Staubli VAL3: PROG.pjx

--- PROG.pjx ---
Parameters version=s7.7.1 stackSize=5000 millimeterUnit=true
Program file=delete.pgx
Program file=deleteItem.pgx
Program file=delEvent.pgx
Program file=duplicate.pgx
Program file=find.pgx
Program file=findItem.pgx
Program file=findTrajItem.pgx
Program file=get.pgx
Program file=getItem.pgx
Program file=getProgItem.pgx
Program file=getSize.pgx
Program file=getSizeItem.pgx
Program file=getType.pgx
Program file=insertItem.pgx
Program file=load.pgx
Program file=loadCycle.pgx
Program file=loadPage.pgx
Program file=new.pgx
Program file=onEdit.pgx
Program file=onInsert.pgx
Program file=onProgEnd.pgx
Program file=onRun.pgx
Program file=onStart.pgx
Program file=onStop.pgx
Program file=pasteItem.pgx
Program file=save.pgx
Program file=scan_prog.pgx
Program file=scanning.pgx
Program file=selectItem.pgx
Program file=setItem.pgx
Program file=showExist.pgx
Program file=unSelectItem.pgx
Program file=write_to_file.pgx
Data file=PROG.dtx
Library alias=saveData path=Disk://saveData/saveData.pjx
Library alias=page path=Disk://kernel/template/page/page.pjx
Library alias=saveProg path=Disk://kernel/template/session/saveProg/PROG/PROG.pjx
Library alias=use path=Disk://kernel/userPage/userPage.pjx
Library alias=language path=Disk://kernel/language/language.pjx
Library alias=cycleStatus path=Disk://cycleStatus/cycleStatus.pjx
Library alias=TrajItem path=Disk://../templates/trajectory/trajectory.pjx
Library alias=sub path=Disk://instruction/SUB/SUB.pjx
Library alias=tcp path=Disk://kernel/tool/tool.pjx
Library alias=saveInputOutput path=Disk://saveInputOutput/saveInputOutput.pjx
Type name=InstrItem path=Disk://kernel/template/InstrItem/InstrItem.pjx
Type name=progItem path=Disk://kernel/template/progItem/progItem.pjx
Type name=TrajectoryItem path=Disk://kernel/template/TrajectoryItem/TrajectoryItem.pjx

--- PROG.dtx ---
num nChar = 89
num nFile = 2
progItem pEdit
  [0]
    InstrItem iEvent[2]
      [0]
        string sType = "PALLET"
        string sData = "prise"
      [1]
        string sType = "OUT"
        string sData = "bOut0>OFF AND bOut1>ON"
    string sID = "pick_place"
public string sItems
string sLine[100]
string sPathTemplate = "Disk://kernel/template/"
string sSession
string sTrajType
public string sWrite

--- delete.pgx ---
public program delete(string x_sName (dimensions=1), num x_nResult (dimensions=1))
  local string l_sItem
  local num l_nDefault
begin
  //
  // delete the select program in
  //
  if isDefined(saveProg:pProg[x_sName])
    // delete
    delete(saveProg:pProg[x_sName])
  endIf
end

--- deleteItem.pgx ---
public program deleteItem(num x_nIndex, num& x_nResult[])
  local num l_nFound
  local num l_nSize
  local num i
  local InstrItem l_sEvent
begin
  //
  // delete the selected field
  //
  call getSizeItem(l_nSize)
  l_nFound=0
  for i=0 to (l_nSize-1)
    call getItem(l_sEvent,i)
    if find(l_sEvent.sType,"#")!=-1
      l_nFound=-1
      call delEvent(i)
      i=i-1
      call getSizeItem(l_nSize)
    endIf
  endFor
  //
  // if there are no marked events delete the select one
  //
  if x_nIndex!=-1 and l_nFound==0
    call delEvent(x_nIndex)
  endIf
end

--- delEvent.pgx ---
program delEvent(num x_nIndex (dimensions=1))
begin
  // delete the item
  if size(pEdit.iEvent)>1
    delete(pEdit.iEvent[x_nIndex])
  else
    pEdit.iEvent.sType=""
    pEdit.iEvent.sData=""
  endIf
end

--- duplicate.pgx ---
public program duplicate(string x_sCopy (dimensions=1), string x_sPaste (dimensions=1), num& x_nResult[] (dimensions=1))
  local num i
  local num l_nSize
  local string l_sItem
  local bool l_bFound
begin
  //
  // return -1 if present
  //
  // create a new one
  call new(x_sPaste,i)
  // duplicate
  saveProg:pProg[x_sPaste]=saveProg:pProg[x_sCopy]
  saveProg:pProg[x_sPaste].sID=x_sPaste
end

--- find.pgx ---
public program find(string& x_sItem[] (dimensions=1), bool& x_bFound[] (dimensions=1))
  local num i
  local num l_nSize
  local string l_sEvent
begin
  // check if the item has been found
  x_bFound=isDefined(saveProg:pProg[x_sItem])
end

--- findItem.pgx ---
public program findItem(InstrItem x_iItem, num& x_nResult[], bool x_bUseSession)
// procedure
  local num i
  local num j
  local num k
  local num l_nSize
  local string l_sProgName
  local bool l_bFound
  local num l_nSizeItem
  local InstrItem l_iItem
  local num z
  local string l_sSession
  local string l_sEmpty
  local string l_sMessage
  local string l_sPath
begin
  //
  // search in all of the program the x_iItem
  //
  // check if the cycle is running or the simulation...
  //
  // mutex the resource
  //
  if !cycleStatus:bCycle and !cycleStatus:bSimulation
    setMutex(cycleStatus:bMutex)
    // save the actual session
    call saveData:getSession(l_sSession)
    // clean the string
    call use:stringCopy(l_sEmpty,sSession)
    if x_bUseSession
      // get the session list
      call saveData:getListSession(sSession)
    endIf
    cls()
    // show the timerDialog
    call use:timerDialog("#",0)
    call use:type(1,2,"SEARCHING: "+x_iItem.sType+" "+x_iItem.sData)
    // for all the session
    for z=0 to size(sSession)-1
      if x_bUseSession
        // scan ALL
        call saveData:changeSession(sSession[z])
      else
        // just the local ONE
        sSession[z]=l_sSession
        z=size(sSession)-1
      endIf
      // look in all the current path
      call getSize(l_nSize)
      for i=0 to (l_nSize-1)
        // load all the program
        call get(l_sProgName,i)
        if l_sProgName!=""
          // SHOW THE program name
          l_sMessage="SESSION:"+sSession[z]+" >PROG "+l_sProgName
          call use:typeLen(1,5,l_sMessage,38)
          // load the select program and search inside
          call load(l_sProgName,x_nResult)
          if x_nResult==0
            // SEARCH IN ALL THE ITEMS
            call getSizeItem(l_nSizeItem)
            if l_nSize!=0
              for j=0 to (l_nSizeItem-1)
                call getItem(l_iItem,j)
                // look inside
                l_bFound=(l_iItem.sType==x_iItem.sType and(l_iItem.sData==x_iItem.sData or find(l_iItem.sData," "+x_iItem.sData)!=-1))
                // use nested items
                if x_iItem.sType=="IN" or x_iItem.sType=="OUT" or x_iItem.sType=="NUM"
                  l_bFound=l_bFound or (find(l_iItem.sData,x_iItem.sType)!=-1 and find(l_iItem.sData," "+x_iItem.sData)!=-1)
                else
                  l_bFound=l_bFound or (find(l_iItem.sData,x_iItem.sType)!=-1 and find(l_iItem.sData+"#"," "+x_iItem.sData+"#")!=-1)
                endIf
                // FOUND IT
                if l_bFound
                  x_nResult=-1
                  call language:message(l_sMessage,23)
                  popUpMsg(l_sMessage+x_iItem.sType+" "+x_iItem.sData+chr(10)+"SESSION:"+sSession[z]+chr(10)+"PROG: "+l_sProgName+" > "+l_iItem.sType+" "+l_iItem.sData)
                  // back
                  call saveData:changeSession(l_sSession)
                  // release
                  cycleStatus:bMutex=false
                  return
                endIf
                delay(0)
              endFor
            endIf
          else
            popUpMsg("error loading...SESSION:"+sSession[z]+">PROG "+l_sProgName+" error "+toString("",x_nResult))
            // release
            cycleStatus:bMutex=false
            return
          endIf
        endIf
        delay(0)
      endFor
      delay(0)
    endFor
    // check if the type is a TRAJ...
    call saveData:getPathInstr(x_iItem.sType,l_sPath)
    if find(l_sPath,"trajectory")==-1
      // SCAN THE SUB
      call sub:findItem(x_iItem,x_nResult,x_bUseSession)
      if x_nResult!=-1
        // SCAN ALL THE TRAJ
        call findTrajItem(x_iItem,x_nResult)
      endIf
      if x_nResult!=-1
        // SCAN ALL THE TCP
        call tcp:findItem(x_iItem,x_nResult)
      endIf
      // back
    endIf
    // set the old session
    call saveData:changeSession(l_sSession)
    // release
    cycleStatus:bMutex=false
  endIf
end

--- findTrajItem.pgx ---
program findTrajItem(InstrItem x_iItem, num& x_nResult)
  local num i
  local string l_sPath
  local num l_nSize
  local num j
  local string l_sItem
  local num l_nSizeItem
  local num k
  local TrajectoryItem l_tTraj
  local num z
  local bool l_bnFound
  local string l_sMessage
  local string l_sSession
  local num l_nResult
  local bool l_bFound
begin
  // scan all the trajectory
  for i=0 to size(saveData:sTrajType)-1
    call saveData:getPathInstr(saveData:sTrajType[i],l_sPath)
    // TRAJECTORY
    l_nResult=TrajItem:libLoad(l_sPath)
    delay(0)
    if l_nResult==0
      call TrajItem:getSize(l_nSize)
      for j=0 to l_nSize-1
        // load the trajectory
        call TrajItem:get(l_sItem,j)
        call saveData:getSession(l_sSession)
        // SHOW THE trajectory name
        l_sMessage="SESSION:"+l_sSession+">"+saveData:sTrajType[i]+" "+l_sItem
        call use:typeLen(1,5,l_sMessage,38)
        call TrajItem:load(l_sItem,x_nResult)
        if x_nResult==0
          call TrajItem:getSizeItem(false,l_nSizeItem)
          // scan for the action
          for k=0 to l_nSizeItem-1
            // get the item
            call TrajItem:getTrajItem(l_tTraj,k)
            // scan deeper for all the action
            for z=0 to size(l_tTraj.iInstr)-1
              // look inside
              l_bFound=(l_tTraj.iInstr[z].sType==x_iItem.sType and(l_tTraj.iInstr[z].sData==x_iItem.sData or find(l_tTraj.iInstr[z].sData,x_iItem.sData+">")!=-1))
              // use nested items
              l_bFound=l_bFound or find(l_tTraj.iInstr[z].sType+" "+l_tTraj.iInstr[z].sData,x_iItem.sData)!=-1
              // FOUND IT
              if l_bFound
                x_nResult=-1
                call language:message(l_sMessage,23)
                popUpMsg(l_sMessage+x_iItem.sType+" "+x_iItem.sData+chr(10)+"SESSION:"+l_sSession+chr(10)+saveData:sTrajType[i]+" "+l_sItem+" > "+l_tTraj.iInstr[z].sType+" "+l_tTraj.iInstr[z].sData)
                // back
                return
              endIf
            endFor
          endFor
        else
          popUpMsg("error loading...SESSION:"+l_sSession+">"+saveData:sTrajType[i]+" "+l_sItem+" error "+toString("",x_nResult))
        endIf
      endFor
    endIf
  endFor
end

--- get.pgx ---
public program get(string& x_sItem[] (dimensions=1), num x_nIndex (dimensions=1))
  local string l_sKey
  local num i
begin
  // start from the first
  l_sKey=first(saveProg:pProg)
  // search it
  while l_sKey!=""
    x_sItem=l_sKey
    l_sKey=next(saveProg:pProg[l_sKey])
    if i==x_nIndex
      return
    else
      i=i+1
    endIf
  endWhile
end

--- getItem.pgx ---
public program getItem(InstrItem& x_sItem (dimensions=1), num x_nIndex (dimensions=1))
begin
  // give back the instruction
  x_sItem=pEdit.iEvent[x_nIndex]
end

--- getProgItem.pgx ---
public program getProgItem(progItem& x_pProgItem, string x_sName)
  local num l_nResult
  local string l_sPath
  local string l_sName
begin
  if isDefined(saveProg:pProg[x_sName])
    // give back
    x_pProgItem=saveProg:pProg[x_sName]
    x_pProgItem.sID=x_sName
  else
    // TODO
    popUpMsg("PROG: "+x_sName+" NOT FOUND ")
    x_pProgItem.sID=""
  endIf
end

--- getSize.pgx ---
public program getSize(num& x_nSize[] (dimensions=1))
  local num i
  local num l_nSize
  local bool l_bFound
  local string l_sEmpty
  local string l_sPath
  local string l_sType
  local string l_sKey
  local string l_sItem
begin
  // give back the size to trajectory field
  x_nSize=size(saveProg:pProg)
end

--- getSizeItem.pgx ---
public program getSizeItem(num& x_nSize[] (dimensions=1))
begin
  // get the size
  if pEdit.iEvent.sType==""
    x_nSize=0
  else
    x_nSize=size(pEdit.iEvent)
  endIf
end

--- getType.pgx ---
program getType(string& x_sType[] (dimensions=1))
  local num l_nPos
  local string l_sPath
begin
  // get the TypePath
  l_sPath=libPath()
  do
    l_nPos=find(l_sPath,"/")
    if l_nPos==-1
      l_nPos=find(l_sPath,"\")
    endIf
    if l_nPos!=-1
      l_sPath=right(l_sPath,len(l_sPath)-l_nPos-1)
    endIf
  until l_nPos==-1
  x_sType=l_sPath
end

--- insertItem.pgx ---
public program insertItem(InstrItem& x_sItem[] (dimensions=1), num x_nIndex (dimensions=1))
  local num l_sItem
begin
  if x_nIndex<=0
    x_nIndex=0
  else
    insert(pEdit.iEvent[x_nIndex])
  endIf
  call setItem(x_sItem,x_nIndex)
end

--- load.pgx ---
public program load(string x_sItem, num& x_nResult[])
  local string l_sPath
  local string l_sName
  local string l_sType
  local progItem l_pNull
  local string l_sMessage
begin
  // check the libPath
  call getType(l_sType)
  // load it
  if find(saveProg:libPath(),saveData:sPathProg)==-1
    x_nResult=saveProg:libLoad(saveData:sPathProg+l_sType)
    delay(0)
    if saveData:bDebug
      ? "loading PROG..."+saveData:sPathProg+l_sType
    endIf
  endIf
  // reload the edit template
  if isDefined(saveProg:pProg[x_sItem].sID) and x_sItem!=""
    // refresh the iD...
    saveProg:pProg[x_sItem].sID=x_sItem
    // update the select item
    pEdit=saveProg:pProg[x_sItem]
  elseIf x_sItem!=""
    // not FOUND
    call language:message(l_sMessage,-7)
    x_nResult=-1
    popUpMsg(l_sMessage+x_sItem)
    // use an empty one
    pEdit.sID=""
  endIf
end

--- loadCycle.pgx ---
public program loadCycle(string x_sItem, num& x_nResult[])
  local string l_sName
  local string l_sPath
  local string l_sType
begin
  call getType(l_sType)
  // load it
  if find(saveProg:libPath(),saveData:sPathProg)==-1
    x_nResult=saveProg:libLoad(saveData:sPathProg+l_sType)
    delay(0)
    if saveData:bDebug
      ? "loading PROG..."+saveData:sPathProg+l_sType
    endIf
    // check if exist or not
  endIf
  // reload the edit template
  if isDefined(saveProg:pProg[x_sItem].sID) and x_sItem!=""
    // refresh the iD...
    saveProg:pProg[x_sItem].sID=x_sItem
    // item found
    x_nResult=0
  endIf
end

--- new.pgx ---
public program new(string x_sName (dimensions=1), num& x_nResult[] (dimensions=1))
  local string l_sMessage
begin
  // new element
  if insert(saveProg:pProg[x_sName])
    saveProg:pProg[x_sName].sID=x_sName
    x_nResult=0
  else
    call language:message(l_sMessage,-2)
    popUpMsg(l_sMessage)
    x_nResult=-1
  endIf
end

--- onEdit.pgx ---
public program onEdit(string& x_sItem[] (dimensions=1))
  local num l_nResult
begin
  //
  // go to the view instruction page
  //
  if size(x_sItem)>1
    call load(x_sItem,l_nResult)
    // give it back
    x_sItem[1]=x_sItem
    x_sItem="Disk://instruction/PROG/page_viewInstr"
  endIf
end

--- onInsert.pgx ---
public program onInsert(string& x_sItem[])
  local string l_sEvent
  local num i
  local num l_nSize
  local string l_sMessage
  local num l_nKey
  local bool l_bFound
begin
  cls()
  call use:setView(false)
  call use:setSizeList(19,0,19,11)
  //
  // Prog
  //
  call use:listcreate("PROG")
  call getSize(l_nSize)
  // refresh the list
  for i=0 to l_nSize-1
    call get(l_sEvent,i)
    if l_sEvent!="" and left(l_sEvent,1)!="#" and l_sEvent!="HOME1" and l_sEvent!="HOME2"
      // check it
      if saveData:sProgFilter!=""
        l_bFound=find(l_sEvent,saveData:sProgFilter)==-1
      else
        l_bFound=true
      endIf
      // add
      if l_bFound
        call use:listadd(l_sEvent)
      endIf
    endIf
  endFor
  // update the list
  call use:listupdate(0)
  call language:message(l_sMessage,60)
  call use:typeLen(0,13,l_sMessage,40)
  do
    l_nKey=get()
    call use:listevent(l_nKey,i,x_sItem)
  until l_nKey==270 or l_nKey==255
  // exit
  if l_nKey==255
    x_sItem=""
  endIf
end

--- onRun.pgx ---
public program onRun(string& x_sItem[] (dimensions=1))
begin
  // PROG NAME x_sItem
  // SET THE CALL SUB..
  cycleStatus:bCALL=true
  if x_sItem!=""
    cycleStatus:iToSuperV.sType="PROG"
    cycleStatus:iToSuperV.sData=x_sItem
  endIf
  use:bUseRefresh=true
end

--- onStart.pgx ---
public program onStart(string& x_sItem[] (dimensions=1))
  local string l_sType
  local num i
  local string l_sPath
  local num l_nResult
  local string l_sName
begin

end

--- onStop.pgx ---
public program onStop(string& x_sItem[])
begin
  if x_sItem=="kill"
    saveProg:libLoad("Disk://kernel/template/session/saveProg/PROG")
    delay(0)
    TrajItem:libLoad("Disk://../templates/trajectory/trajectory.pjx")
    delay(0)
  endIf
end

--- pasteItem.pgx ---
public program pasteItem(num& x_nIndex[] (dimensions=1))
  local num l_nSize
  local num i
  local InstrItem l_sItem
  local num l_nTemp
  local string l_sRight
begin
  call getSizeItem(l_nSize)
  l_nTemp=x_nIndex+1
  for i=0 to (l_nSize-1)
    call getItem(l_sItem,i)
    if find(l_sItem.sType,"#")!=-1
      if l_nTemp<=i
        i=i+1
      endIf
      l_sItem.sType=right(l_sItem.sType,len(l_sItem.sType)-1)
      call insertItem(l_sItem,l_nTemp)
      l_nTemp=l_nTemp+1
      l_nSize=l_nSize+1
    endIf
  endFor
  // unselect all
  call unSelectItem()
end

--- save.pgx ---
public program save(string x_sName, num& x_nResult[])
begin
  // save it
  if isDefined(saveProg:pProg[pEdit.sID])
    saveProg:pProg[pEdit.sID]=pEdit
  endIf
  x_nResult=saveProg:libSave()
end

--- scan_prog.pgx ---
public program scan_prog(string x_sProg (dimensions=1), string x_sName (dimensions=1))
  local string l_sEmpty
  local num l_nId
begin
  // do the scan and save the file
  // init the sWrite
  call use:stringCopy(l_sEmpty,sWrite)
  // open the file
  nFile=$fileOpen(x_sName+".txt","w")
  // start the scanning
  l_nId=0
  call scanning(x_sProg,0,l_nId,false)
  // save the file
  $fileSet(nFile,sWrite,size(sWrite))
  $fileClose(nFile)
end

--- scanning.pgx ---
public program scanning(string x_sProgram, num x_nX, num& x_nY[], bool x_bSaveResult)
  local string l_sProgram
  local string l_sEmpty
  local string l_sItem[100]
  local string l_sMinus
  local string l_sLine[5]
  local string l_sTrajName
  local num i
  local num l_nSize
  local num l_nPos
  local num j
  local num l_nLine
  local num k
  local InstrItem l_iItem
  local string l_sPath
  local num l_nSizeItem
  local num l_nResult
  local progItem l_pProg
  local TrajectoryItem l_tTraj
begin
  //
  // open the program
  //
  call load(x_sProgram,i)
  if i==0
    //
    // get the item
    //
    call getSizeItem(l_nSize)
    //
    // print all the line
    //
    for i=0 to l_nSize-1
      //
      // init the local variable
      //
      l_sEmpty=""
      l_sMinus=""
      l_sProgram=""
      for j=0 to size(l_sLine)-1
        l_sLine[j]=""
      endFor
      l_nLine=0
      //
      // scan the item looking for some tray type or SUB
      //
      call getItem(l_iItem,i)
      // find if there is a program inside
      if l_iItem.sType=="PROG"
        // find the program name
        l_sProgram=l_iItem.sData
      elseIf l_iItem.sType=="IF"
        // scan for the IF
        l_nPos=find(l_iItem.sData,"PROG ")
        if l_nPos!=-1
          // find the program name
          l_sProgram=right(l_iItem.sData,len(l_iItem.sData)-l_nPos-len("PROG "))
        endIf
      endIf
      call saveInputOutput:replaceIO(l_iItem.sData,l_iItem.sType,l_iItem.sData)
      l_sItem[i]=l_iItem.sType+" "+l_iItem.sData
      //
      // set the string in a nChar + 1 space
      //
      if len(l_sItem[i])>nChar
        // save the line
        l_nLine=roundUp(len(l_sItem[i])/(nChar-1))-1
        for j=0 to l_nLine
          if j==0
            // FIRST LINE
            // divide it
            l_sLine[j]=left(l_sItem[i],(nChar-1))
            // cut it
            if len(l_sLine[j])==(nChar-1)
              l_sLine[j]=l_sLine[j]+"~ "
              l_sItem[i]=right(l_sItem[i],len(l_sItem[i])-(nChar-1))
            endIf
          else
            // OTHERS LINE
            // divide it
            l_sLine[j]="-"+left(l_sItem[i],(nChar-2))
            // cut it
            if len(l_sLine[j])==(nChar-1)
              l_sLine[j]=l_sLine[j]+"~ "
              l_sItem[i]=right(l_sItem[i],len(l_sItem[i])-(nChar-2))
            endIf
          endIf
        endFor
      else
        // set the string
        l_sLine=l_sItem[i]
      endIf
      if len(l_sLine[l_nLine])<(nChar+1)
        for j=0 to (nChar-len(l_sLine[l_nLine]))
          // fill the empty
          l_sEmpty=l_sEmpty+" "
        endFor
      endIf
      // look if there is a program to write
      if l_sProgram!=""
        // write the line
        for j=0 to l_nLine
          if j==l_nLine
            // write the minus
            call write_to_file(x_nX,x_nY,l_sLine[j],true)
          else
            // write full sentence
            call write_to_file(x_nX,x_nY,l_sLine[j],false)
            x_nY=x_nY+1
          endIf
        endFor
        // scan again
        x_nY=x_nY+1
        call scanning(l_sProgram,x_nX+15,x_nY,x_bSaveResult)
        // recover the last program
        call load(x_sProgram,i)
      else
        // write the line
        for j=0 to l_nLine
          if j==l_nLine
            // write the space
            call write_to_file(x_nX,x_nY,l_sLine[j]+l_sEmpty,false)
          else
            // no space
            call write_to_file(x_nX,x_nY,l_sLine[j],false)
          endIf
          x_nY=x_nY+1
        endFor
        // get inside the trajectory field
        call saveData:getPathInstr(l_iItem.sType,l_sPath)
        // TRAJECTORY
        if TrajItem:libLoad(l_sPath)==0
          delay(0)
          // scan for the action
          call TrajItem:load(l_iItem.sData,l_nResult)
          call TrajItem:getSizeItem(false,l_nSizeItem)
          // patch for the pallet
          if l_iItem.sType=="PALLET"
            l_nSizeItem=1
          endIf
          for j=0 to l_nSizeItem-1
            // get the item
            call TrajItem:getTrajItem(l_tTraj,j)
            // scan for the TCP
            if l_tTraj.nTcpAction==1
              call write_to_file(x_nX,x_nY,"   -TCP ON ",false)
              //add one line
              x_nY=x_nY+1
            elseIf l_tTraj.nTcpAction==2
              call write_to_file(x_nX,x_nY,"   -TCP OFF",false)
              //add one line
              x_nY=x_nY+1
            endIf
            for k=0 to size(l_tTraj.iInstr)-1
              if l_tTraj.iInstr[k].sType!=""
                call saveInputOutput:replaceIO(l_tTraj.iInstr[k].sData,l_tTraj.iInstr[k].sType,l_tTraj.iInstr[k].sData)
                call write_to_file(x_nX,x_nY,"   -"+l_tTraj.iInstr[k].sType+" "+l_tTraj.iInstr[k].sData,false)
                //add one line
                x_nY=x_nY+1
                if l_tTraj.iInstr[k].sType=="SUB"
                  // SUB
                  call sub:getProgItem(l_pProg,l_tTraj.iInstr[k].sData)
                  l_nSizeItem=size(l_pProg.iEvent)
                  for j=0 to l_nSizeItem-1
                    if l_pProg.iEvent[j].sType!=""
                      call saveInputOutput:replaceIO(l_pProg.iEvent[j].sData,l_pProg.iEvent[j].sType,l_pProg.iEvent[j].sData)
                      call write_to_file(x_nX,x_nY,"        "+l_pProg.iEvent[j].sType+" "+l_pProg.iEvent[j].sData,false)
                      //add one line
                      x_nY=x_nY+1
                    endIf
                  endFor
                endIf
              endIf
            endFor
          endFor
        elseIf l_iItem.sType=="SUB"
          // SUB
          call sub:getProgItem(l_pProg,l_iItem.sData)
          l_nSizeItem=size(l_pProg.iEvent)
          for j=0 to l_nSizeItem-1
            if l_pProg.iEvent[j].sType!=""
              call saveInputOutput:replaceIO(l_pProg.iEvent[j].sData,l_pProg.iEvent[j].sType,l_pProg.iEvent[j].sData)
              call write_to_file(x_nX,x_nY,"    "+l_pProg.iEvent[j].sType+" "+l_pProg.iEvent[j].sData,false)
              //add one line
              x_nY=x_nY+1
            endIf
          endFor
        endIf
      endIf
      delay(0)
    endFor
  endIf
end

--- selectItem.pgx ---
public program selectItem(num x_nIndex (dimensions=1))
  local InstrItem l_sItem
begin
  //
  // select or unselect one item
  //
  call getItem(l_sItem,x_nIndex)
  if find(l_sItem.sType,"#")==-1
    l_sItem.sType="#"+l_sItem.sType
  else
    l_sItem.sType=right(l_sItem.sType,len(l_sItem.sType)-1)
  endIf
  // set Item
  call setItem(l_sItem,x_nIndex)
end

--- setItem.pgx ---
public program setItem(InstrItem& x_sItem[] (dimensions=1), num& x_nIndex[] (dimensions=1))
begin
  // set IT
  pEdit.iEvent[x_nIndex]=x_sItem
end

--- unSelectItem.pgx ---
public program unSelectItem()
  local InstrItem l_sEvent
  local num i
  local num l_nSize
begin
  // deselect all
  call getSizeItem(l_nSize)
  for i=0 to (l_nSize-1)
    call getItem(l_sEvent,i)
    if find(l_sEvent.sType,"#")!=-1
      l_sEvent.sType=right(l_sEvent.sType,len(l_sEvent.sType)-1)
      call setItem(l_sEvent,i)
    endIf
  endFor
end

--- write_to_file.pgx ---
program write_to_file(num x_nX (dimensions=1), num x_nY (dimensions=1), string x_sItem (dimensions=1), bool x_bCall (dimensions=1))
  local num i
  local num l_nSize
  local string l_sFill
begin
  //
  // check the size
  //
  l_nSize=size(sWrite)-x_nY
  if l_nSize<=0
    for i=0 to abs(l_nSize)
      // insert new Line
      insert(sWrite[size(sWrite)])
    endFor
  endIf
  //
  // write in the line
  //
  // test if the len is ok
  //
  l_nSize=len(sWrite[x_nY])-x_nX
  if l_nSize<=0
    for i=0 to abs(l_nSize)
      // insert white space if the item on the left is a PROG
      sWrite[x_nY]=insert(sWrite[x_nY]," ",len(sWrite[x_nY]))
    endFor
    // insert the line
    sWrite[x_nY]=replace(sWrite[x_nY],x_sItem,0,x_nX)
  else
    if x_bCall
      //need to insert for all the line an empty string of nChar
      for i=0 to size(sWrite)-1
        call use:strfill(l_sFill,nChar+1,l_sFill)
        //        if (mid(sWrite[i],1,x_nX+nChar)=="═")
        //          call use:strfillchr(l_sFill,l_sFill,"═")
        //          // line
        //          sWrite[i]=insert(sWrite[i],l_sFill,x_nX+nChar+1)
        //        else
        // space
        sWrite[i]=insert(sWrite[i],l_sFill,x_nX+nChar+1)
        //       endIf
      endFor
    endIf
    // replace the string
    sWrite[x_nY]=replace(sWrite[x_nY],x_sItem,nChar+1,x_nX)
  endIf
end
